FUNCTION_BLOCK FB_PipelineConsumer
VAR
    stage : B4Pipeline_Plc.FB_PipelineStage;
    bStageError : BOOL;
END_VAR

stage(value := -1);
bStageError := stage.bError;

END_FUNCTION_BLOCK

(* stored: Version 1.1.0.1
   POU FB_PipelineConsumer: Id {055d9f00-73cd-4e40-a382-ce6caa376910}, SpecialFunc None *)
